TYPE ST_KeyenceLaser_Command_Request_Completion_Clear :
STRUCT
Command_Request_Complete_Clear		: BIT;
Reserve_0							: BIT;
Reserve_1							: BIT;
Reserve_2							: BIT;
Reserve_3							: BIT;
Reserve_4							: BIT;
Reserve_5							: BIT;
Reserve_6							: BIT;
END_STRUCT
END_TYPE

(* stored: Version 1.1.0.1, ProductVersion 3.1.4024.11
   DUT ST_KeyenceLaser_Command_Request_Completion_Clear: Id {c38b2002-8bdf-47e3-b611-f704388f7f3f} *)
